TYPE udt_IV2_Outputs :
STRUCT
	Program_Switch_RQST:BOOL;
	Trigger_RQST:BOOL;
	Master_Image_RQST:BOOL;
	SD_Save_Stop_RQST:BOOL;
	Reset_Statistics_RQST:BOOL;
	Error_Clear_RQST:BOOL;
	ProgramNum:ARRAY[0..3] OF BOOL;
END_STRUCT
END_TYPE

(* stored: Version 1.1.0.1, ProductVersion 3.1.4024.12
   DUT udt_IV2_Outputs: Id {ce48f901-b81a-44c7-8fbe-741450114800} *)
